{attribute 'qualified_only'}
{attribute 'strict'}
TYPE E_NOTT_CRYO_CTRL_STATE :
(
	NONE 			:= 0,
	WARM_PRESS,				// Warm & Pressurized
	WARM_VACUUM,			// Warm & Vacuum
	COOLING_DOWN,			// Cooling down
	COLD,					// Cold, i.e. fully operational
	WARMING_UP,				// Warming up
	ERROR					// Controller failure
);
END_TYPE

(* stored: Version 1.1.0.1, ProductVersion 3.1.4026.18
   DUT E_NOTT_CRYO_CTRL_STATE: Id {8481a251-a855-4d51-b613-73faf0fd853f} *)
